{attribute 'linkalways'} 
{attribute 'no_explicit_call' := 'This FB is a CLASS and must be accessed using methods or properties'}
{attribute 'enable_dynamic_creation'}
FUNCTION_BLOCK Node_F_VN_NormalizeImageForDisplay EXTENDS VisionNode
VAR
    ipSrcImage : _ITcVnImage;
    ipDestImage : _ITcVnImage;
    eSignedNormalization : _ETcVnSignedNormalization(ETcVnSignedNormalization.TCVN_SN_FIX_ZERO);
    hrPrev : _HRESULT(S_OK);
	hresult : _HRESULT(S_OK);
END_VAR

METHOD PUBLIC  Clone : I_Node
VAR
	pNode : POINTER TO Node_F_VN_NormalizeImageForDisplay;
END_VAR
pNode := __NEW(Node_F_VN_NormalizeImageForDisplay);
Clone := pNode^;
END_METHOD

METHOD FB_init : BOOL
VAR_INPUT
	bInitRetains : BOOL; // if TRUE, the retain variables are initialized (warm start / cold start)
	bInCopyCode : BOOL;  // if TRUE, the instance afterwards gets moved into the copy code (online change)
END_VAR
AddInput('ipSrcImage', ipSrcImage);
AddInput('hrPrev', hrPrev);
AddParameter('eSignedNormalization', eSignedNormalization);
AddOutput('ipDestImage', ipDestImage);
AddOutput('hresult',hresult);
END_METHOD

METHOD PROTECTED OnExecute
hresult.Value := F_VN_NormalizeImageForDisplay(
    ipSrcImage := ipSrcImage.Value,
	ipDestImage := ipDestImage.Value,
    eSignedNormalization := eSignedNormalization.Value,
	hrPrev:= hrPrev.Value);
END_METHOD

METHOD PUBLIC PreExecutionCheck
VAR_INPUT
	Check : I_PreExecutionChecks;
END_VAR
Check.IsTrue(ipSrcImage.IsValid, 'ipSrcImage must contain an image');
END_METHOD

END_FUNCTION_BLOCK

(* stored: Version 1.1.0.1, ProductVersion 3.1.4024.13
   POU Node_F_VN_NormalizeImageForDisplay: Id {336333f5-00e3-07f2-2518-6cd592b85be0}, SpecialFunc None
   Folder Constructor: Id {49af2cda-f980-034d-13b5-e02d1c60426c}
   Method Clone: Id {9cedaec8-e319-04c8-3a5d-c56eec866d5f}
   Method FB_init: Id {61aa1deb-38f7-0c2f-1027-09fb8d1f4350}
   Method OnExecute: Id {9db1a553-05a3-0e2a-3461-fc3a23eb361d}
   Method PreExecutionCheck: Id {d12505d8-7bc9-098f-171d-37f6d1c6edcf} *)
